{attribute 'GeneratedUsingTerminal: KL2531'}
{attribute addProperty BoxType "KL2531"}
{attribute addProperty Id "StatusAT %I*USINT0PositionAT %I*UINT0ExtStatusAT %I*UINT0CtrlAT %Q*USINT0VelocityAT %Q*INT0ExtCtrlAT %Q*UINT0"}
{attribute addProperty CRC "4272151544"}
{attribute addProperty Size "0"}
TYPE Channel_FEA3DBF8 :
STRUCT
	{attribute addProperty Name "Status"}
	Status AT %I* : USINT;
	{attribute addProperty Name "Position"}
	Position AT %I* : UINT;
	{attribute addProperty Name "ExtStatus"}
	ExtStatus AT %I* : UINT;
	{attribute addProperty Name "Ctrl"}
	Ctrl AT %Q* : USINT;
	{attribute addProperty Name "Velocity"}
	Velocity AT %Q* : INT;
	{attribute addProperty Name "ExtCtrl"}
	ExtCtrl AT %Q* : UINT;
END_STRUCT
END_TYPE

(* stored: Version 1.2.0.0, ProductVersion 3.1.4024.9
   DUT Channel_FEA3DBF8: Id {2e57f13a-8000-486f-a662-fea98c9837a7} *)
